// TIA Portal V17 export
// export: Created 2024-08-29T18:23:45.9111074Z, ExportSetting WithDefaults, DisplayName Totally Integrated Automation Portal, DisplayVersion V17 Update 7, DisplayName TIA Portal Openness, DisplayVersion V17 Update 7, DisplayName TIA Portal Version Control Interface, DisplayVersion V17, DisplayName SINAMICS Startdrive Advanced, DisplayVersion V17 SP2, DisplayName SINAMICS Startdrive G110M, G120, G120C, G120D, G120P, G115D, DisplayVersion V17 SP2, DisplayName SINAMICS Startdrive G130, G150, S120, S150, SINAMICS MV, S210, DisplayVersion V17 SP2, DisplayName STEP 7 Professional, DisplayVersion V17 Update 7, DisplayName STEP 7 Safety, DisplayVersion V17 Update 6, DisplayName WinCC Advanced / Unified PC, DisplayVersion V17 Update 7
FUNCTION "stationAlarms" : Void   // FC2, LAD
{ S7_Optimized_Access := 'TRUE' }
VERSION : 0.1
// stored: AutoNumber true, IsIECCheckEnabled false, SetENOAutomatically false, UDAEnableTagReadback false
   VAR_TEMP
      visualizationDefault : Bool;
   END_VAR
   VAR_TEMP   // added for the SCL form of the ladder/FBD networks
      _w1 : Bool;
      _w2 : Bool;
      _w3 : Bool;
      _w4 : Bool;
      _w5 : Bool;
   END_VAR
BEGIN

REGION Network 1: Visualization Defaults
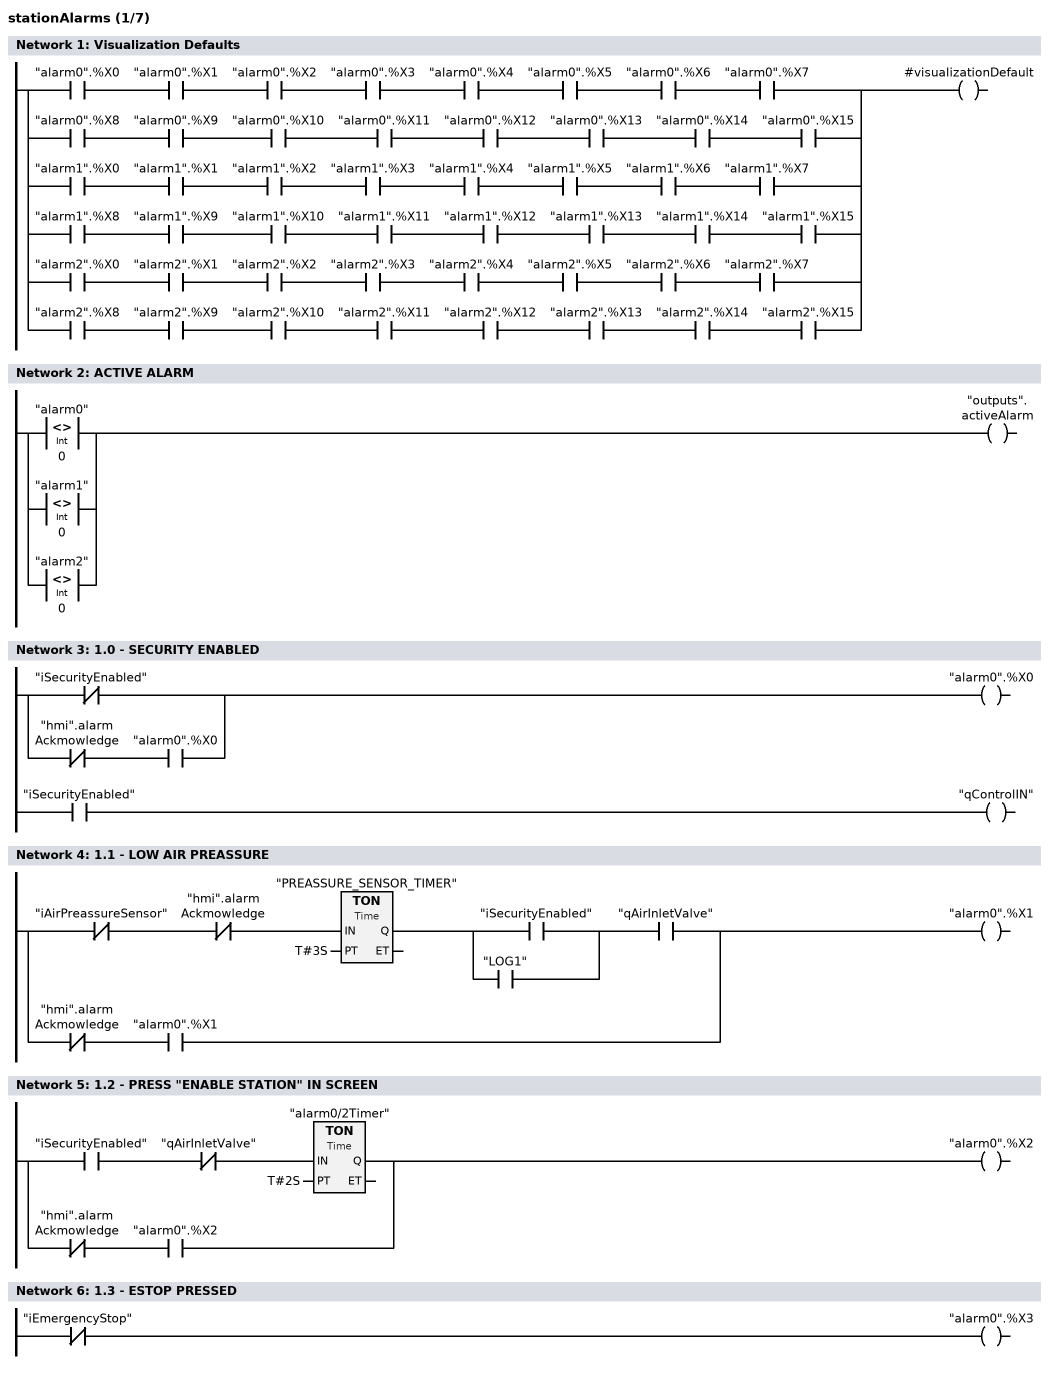
   RUNG wire#powerrail
      Contact( "alarm0".%X0 )
      Contact( "alarm0".%X1 )
      Contact( "alarm0".%X2 )
      Contact( "alarm0".%X3 )
      Contact( "alarm0".%X4 )
      Contact( "alarm0".%X5 )
      Contact( "alarm0".%X6 )
      Contact( "alarm0".%X7 )
      wire#w1
      Coil( #visualizationDefault )
   END_RUNG
   RUNG wire#powerrail
      Contact( "alarm0".%X8 )
      Contact( "alarm0".%X9 )
      Contact( "alarm0".%X10 )
      Contact( "alarm0".%X11 )
      Contact( "alarm0".%X12 )
      Contact( "alarm0".%X13 )
      Contact( "alarm0".%X14 )
      Contact( "alarm0".%X15 )
   END_RUNG wire#w1
   RUNG wire#powerrail
      Contact( "alarm1".%X0 )
      Contact( "alarm1".%X1 )
      Contact( "alarm1".%X2 )
      Contact( "alarm1".%X3 )
      Contact( "alarm1".%X4 )
      Contact( "alarm1".%X5 )
      Contact( "alarm1".%X6 )
      Contact( "alarm1".%X7 )
   END_RUNG wire#w1
   RUNG wire#powerrail
      Contact( "alarm1".%X8 )
      Contact( "alarm1".%X9 )
      Contact( "alarm1".%X10 )
      Contact( "alarm1".%X11 )
      Contact( "alarm1".%X12 )
      Contact( "alarm1".%X13 )
      Contact( "alarm1".%X14 )
      Contact( "alarm1".%X15 )
   END_RUNG wire#w1
   RUNG wire#powerrail
      Contact( "alarm2".%X0 )
      Contact( "alarm2".%X1 )
      Contact( "alarm2".%X2 )
      Contact( "alarm2".%X3 )
      Contact( "alarm2".%X4 )
      Contact( "alarm2".%X5 )
      Contact( "alarm2".%X6 )
      Contact( "alarm2".%X7 )
   END_RUNG wire#w1
   RUNG wire#powerrail
      Contact( "alarm2".%X8 )
      Contact( "alarm2".%X9 )
      Contact( "alarm2".%X10 )
      Contact( "alarm2".%X11 )
      Contact( "alarm2".%X12 )
      Contact( "alarm2".%X13 )
      Contact( "alarm2".%X14 )
      Contact( "alarm2".%X15 )
   END_RUNG wire#w1
   // the same network as SCL:
   #visualizationDefault := ("alarm0".%X0 AND "alarm0".%X1 AND "alarm0".%X2 AND "alarm0".%X3 AND "alarm0".%X4 AND "alarm0".%X5 AND "alarm0".%X6 AND "alarm0".%X7) OR ("alarm0".%X8 AND "alarm0".%X9 AND "alarm0".%X10 AND "alarm0".%X11 AND "alarm0".%X12 AND "alarm0".%X13 AND "alarm0".%X14 AND "alarm0".%X15) OR ("alarm1".%X0 AND "alarm1".%X1 AND "alarm1".%X2 AND "alarm1".%X3 AND "alarm1".%X4 AND "alarm1".%X5 AND "alarm1".%X6 AND "alarm1".%X7) OR ("alarm1".%X8 AND "alarm1".%X9 AND "alarm1".%X10 AND "alarm1".%X11 AND "alarm1".%X12 AND "alarm1".%X13 AND "alarm1".%X14 AND "alarm1".%X15) OR ("alarm2".%X0 AND "alarm2".%X1 AND "alarm2".%X2 AND "alarm2".%X3 AND "alarm2".%X4 AND "alarm2".%X5 AND "alarm2".%X6 AND "alarm2".%X7) OR ("alarm2".%X8 AND "alarm2".%X9 AND "alarm2".%X10 AND "alarm2".%X11 AND "alarm2".%X12 AND "alarm2".%X13 AND "alarm2".%X14 AND "alarm2".%X15);
END_REGION

REGION Network 2: ACTIVE ALARM
   RUNG wire#powerrail
      { S7_Templates := "SrcType := Int" } NE_Contact(in1 := "alarm0", in2 := 0)
      wire#w1
      Coil( "outputs".activeAlarm )
   END_RUNG
   RUNG wire#powerrail
      { S7_Templates := "SrcType := Int" } NE_Contact(in1 := "alarm1", in2 := 0)
   END_RUNG wire#w1
   RUNG wire#powerrail
      { S7_Templates := "SrcType := Int" } NE_Contact(in1 := "alarm2", in2 := 0)
   END_RUNG wire#w1
   // the same network as SCL:
   "outputs".activeAlarm := ("alarm0" <> 0) OR ("alarm1" <> 0) OR ("alarm2" <> 0);
END_REGION

REGION Network 3: 1.0 - SECURITY ENABLED
   RUNG wire#powerrail
      I_Contact( "iSecurityEnabled" )
      wire#w1
      Coil( "alarm0".%X0 )
   END_RUNG
   RUNG wire#powerrail
      I_Contact( "hmi".alarmAckmowledge )
      Contact( "alarm0".%X0 )
   END_RUNG wire#w1
   RUNG wire#powerrail
      Contact( "iSecurityEnabled" )
      Coil( "qControlIN" )
   END_RUNG
   // the same network as SCL:
   "alarm0".%X0 := NOT "iSecurityEnabled" OR (NOT "hmi".alarmAckmowledge AND "alarm0".%X0);
   "qControlIN" := "iSecurityEnabled";
END_REGION

REGION Network 4: 1.1 - LOW AIR PREASSURE
   RUNG wire#powerrail
      I_Contact( "iAirPreassureSensor" )
      I_Contact( "hmi".alarmAckmowledge )
      { S7_Templates := "time_type := Time" } "PREASSURE_SENSOR_TIMER".TON(pt := T#3S, et =>)
      wire#w1
      Contact( "iSecurityEnabled" )
      wire#w2
      Contact( "qAirInletValve" )
      wire#w3
      Coil( "alarm0".%X1 )
   END_RUNG
   RUNG wire#w1
      Contact( "LOG1" )
   END_RUNG wire#w2
   RUNG wire#powerrail
      I_Contact( "hmi".alarmAckmowledge )
      Contact( "alarm0".%X1 )
   END_RUNG wire#w3
   // the same network as SCL:
   "PREASSURE_SENSOR_TIMER".TON(IN := NOT "iAirPreassureSensor" AND NOT "hmi".alarmAckmowledge, PT := T#3S);
   "alarm0".%X1 := ("PREASSURE_SENSOR_TIMER".Q AND ("iSecurityEnabled" OR "LOG1") AND "qAirInletValve") OR (NOT "hmi".alarmAckmowledge AND "alarm0".%X1);
END_REGION

REGION Network 5: 1.2 - PRESS "ENABLE STATION" IN SCREEN
   RUNG wire#powerrail
      Contact( "iSecurityEnabled" )
      I_Contact( "qAirInletValve" )
      { S7_Templates := "time_type := Time" } "alarm0/2Timer".TON(pt := T#2S, et =>)
      wire#w1
      Coil( "alarm0".%X2 )
   END_RUNG
   RUNG wire#powerrail
      I_Contact( "hmi".alarmAckmowledge )
      Contact( "alarm0".%X2 )
   END_RUNG wire#w1
   // the same network as SCL:
   "alarm0/2Timer".TON(IN := "iSecurityEnabled" AND NOT "qAirInletValve", PT := T#2S);
   "alarm0".%X2 := "alarm0/2Timer".Q OR (NOT "hmi".alarmAckmowledge AND "alarm0".%X2);
END_REGION

REGION Network 6: 1.3 - ESTOP PRESSED
   RUNG wire#powerrail
      I_Contact( "iEmergencyStop" )
      Coil( "alarm0".%X3 )
   END_RUNG
   // the same network as SCL:
   "alarm0".%X3 := NOT "iEmergencyStop";
END_REGION

REGION Network 7: 1.4 - MANUAL COMMAND OUT OF MANUAL MODE
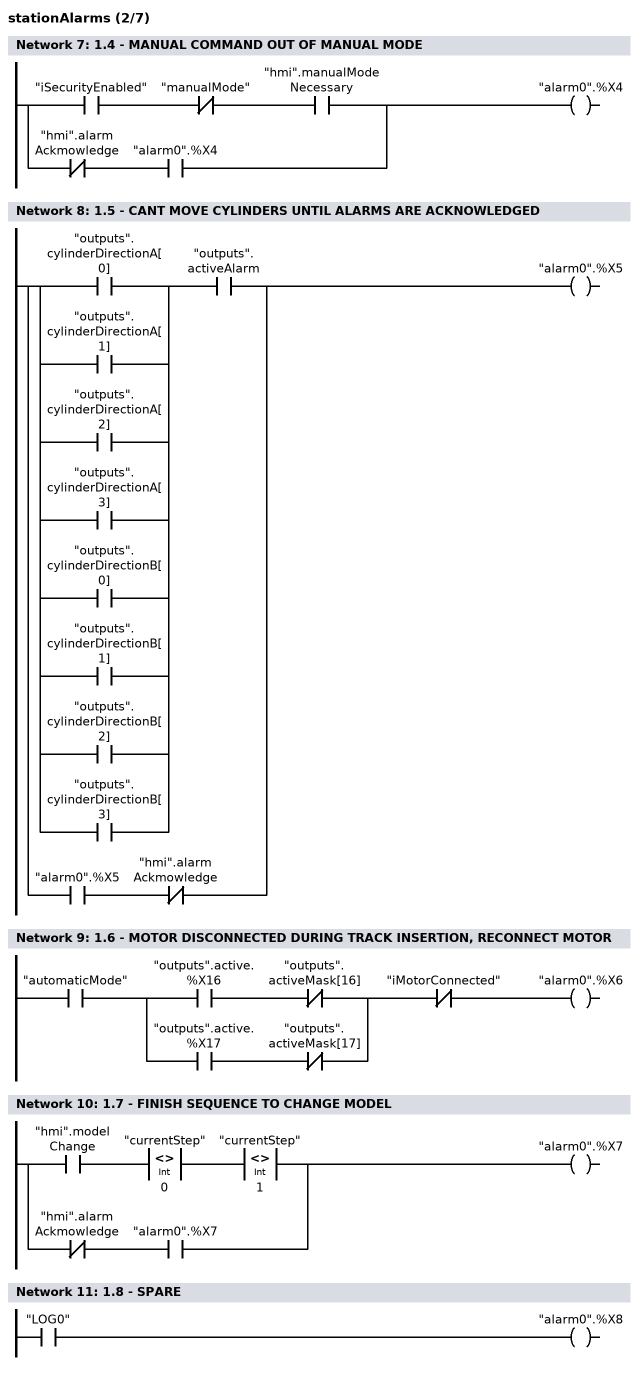
   RUNG wire#powerrail
      Contact( "iSecurityEnabled" )
      I_Contact( "manualMode" )
      Contact( "hmi".manualModeNecessary )
      wire#w1
      Coil( "alarm0".%X4 )
   END_RUNG
   RUNG wire#powerrail
      I_Contact( "hmi".alarmAckmowledge )
      Contact( "alarm0".%X4 )
   END_RUNG wire#w1
   // the same network as SCL:
   "alarm0".%X4 := ("iSecurityEnabled" AND NOT "manualMode" AND "hmi".manualModeNecessary) OR (NOT "hmi".alarmAckmowledge AND "alarm0".%X4);
END_REGION

REGION Network 8: 1.5 - CANT MOVE CYLINDERS UNTIL ALARMS ARE ACKNOWLEDGED
   RUNG wire#powerrail
      Contact( "outputs".cylinderDirectionA[0] )
      wire#w1
      Contact( "outputs".activeAlarm )
      wire#w2
      Coil( "alarm0".%X5 )
   END_RUNG
   RUNG wire#powerrail
      Contact( "outputs".cylinderDirectionA[1] )
   END_RUNG wire#w1
   RUNG wire#powerrail
      Contact( "outputs".cylinderDirectionA[2] )
   END_RUNG wire#w1
   RUNG wire#powerrail
      Contact( "outputs".cylinderDirectionA[3] )
   END_RUNG wire#w1
   RUNG wire#powerrail
      Contact( "outputs".cylinderDirectionB[0] )
   END_RUNG wire#w1
   RUNG wire#powerrail
      Contact( "outputs".cylinderDirectionB[1] )
   END_RUNG wire#w1
   RUNG wire#powerrail
      Contact( "outputs".cylinderDirectionB[2] )
   END_RUNG wire#w1
   RUNG wire#powerrail
      Contact( "outputs".cylinderDirectionB[3] )
   END_RUNG wire#w1
   RUNG wire#powerrail
      Contact( "alarm0".%X5 )
      I_Contact( "hmi".alarmAckmowledge )
   END_RUNG wire#w2
   // the same network as SCL:
   "alarm0".%X5 := (("outputs".cylinderDirectionA[0] OR "outputs".cylinderDirectionA[1] OR "outputs".cylinderDirectionA[2] OR "outputs".cylinderDirectionA[3] OR "outputs".cylinderDirectionB[0] OR "outputs".cylinderDirectionB[1] OR "outputs".cylinderDirectionB[2] OR "outputs".cylinderDirectionB[3]) AND "outputs".activeAlarm) OR ("alarm0".%X5 AND NOT "hmi".alarmAckmowledge);
END_REGION

REGION Network 9: 1.6 - MOTOR DISCONNECTED DURING TRACK INSERTION, RECONNECT MOTOR
   RUNG wire#powerrail
      Contact( "automaticMode" )
      wire#w1
      Contact( "outputs".active.%X16 )
      I_Contact( "outputs".activeMask[16] )
      wire#w2
      I_Contact( "iMotorConnected" )
      Coil( "alarm0".%X6 )
   END_RUNG
   RUNG wire#w1
      Contact( "outputs".active.%X17 )
      I_Contact( "outputs".activeMask[17] )
   END_RUNG wire#w2
   // the same network as SCL:
   "alarm0".%X6 := "automaticMode" AND (("outputs".active.%X16 AND NOT "outputs".activeMask[16]) OR ("outputs".active.%X17 AND NOT "outputs".activeMask[17])) AND NOT "iMotorConnected";
END_REGION

REGION Network 10: 1.7 - FINISH SEQUENCE TO CHANGE MODEL
   RUNG wire#powerrail
      Contact( "hmi".modelChange )
      { S7_Templates := "SrcType := Int" } NE_Contact(in1 := "currentStep", in2 := 0)
      { S7_Templates := "SrcType := Int" } NE_Contact(in1 := "currentStep", in2 := 1)
      wire#w1
      Coil( "alarm0".%X7 )
   END_RUNG
   RUNG wire#powerrail
      I_Contact( "hmi".alarmAckmowledge )
      Contact( "alarm0".%X7 )
   END_RUNG wire#w1
   // the same network as SCL:
   "alarm0".%X7 := ("hmi".modelChange AND ("currentStep" <> 0) AND ("currentStep" <> 1)) OR (NOT "hmi".alarmAckmowledge AND "alarm0".%X7);
END_REGION

REGION Network 11: 1.8 - SPARE
   RUNG wire#powerrail
      Contact( "LOG0" )
      Coil( "alarm0".%X8 )
   END_RUNG
   // the same network as SCL:
   "alarm0".%X8 := "LOG0";
END_REGION

REGION Network 12: 1.9 - WRONG TAG
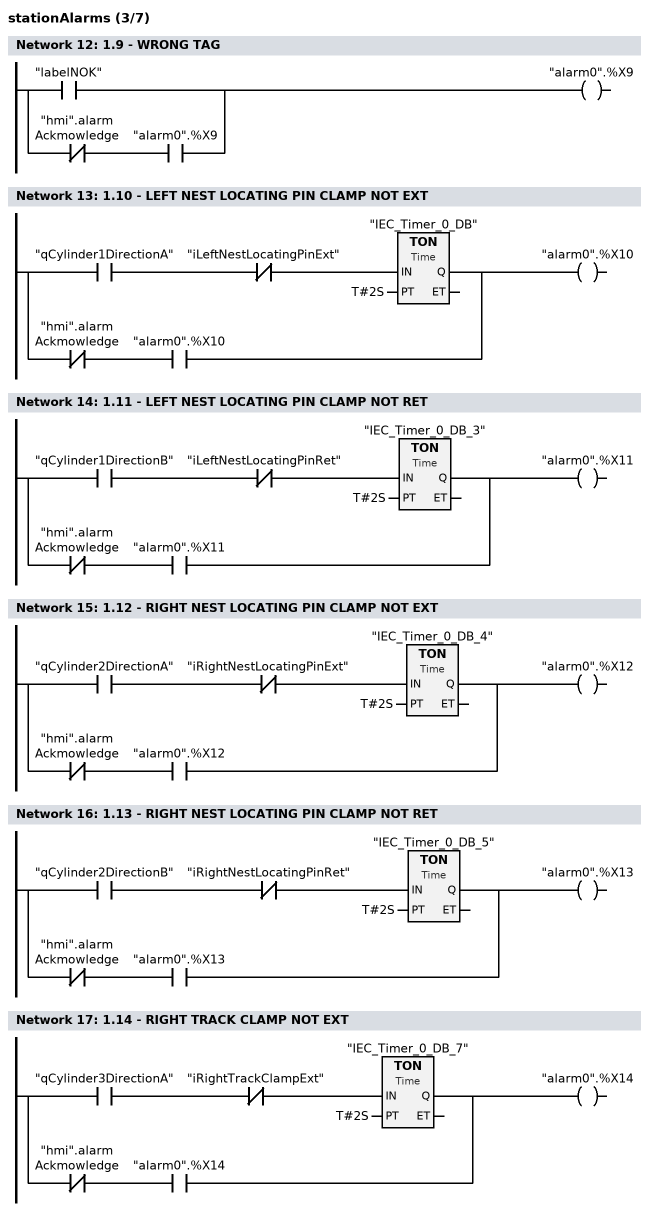
   RUNG wire#powerrail
      Contact( "labelNOK" )
      wire#w1
      Coil( "alarm0".%X9 )
   END_RUNG
   RUNG wire#powerrail
      I_Contact( "hmi".alarmAckmowledge )
      Contact( "alarm0".%X9 )
   END_RUNG wire#w1
   // the same network as SCL:
   "alarm0".%X9 := "labelNOK" OR (NOT "hmi".alarmAckmowledge AND "alarm0".%X9);
END_REGION

REGION Network 13: 1.10 - LEFT NEST LOCATING PIN CLAMP NOT EXT
   RUNG wire#powerrail
      Contact( "qCylinder1DirectionA" )
      I_Contact( "iLeftNestLocatingPinExt" )
      { S7_Templates := "time_type := Time" } "IEC_Timer_0_DB".TON(pt := T#2S, et =>)
      wire#w1
      Coil( "alarm0".%X10 )
   END_RUNG
   RUNG wire#powerrail
      I_Contact( "hmi".alarmAckmowledge )
      Contact( "alarm0".%X10 )
   END_RUNG wire#w1
   // the same network as SCL:
   "IEC_Timer_0_DB".TON(IN := "qCylinder1DirectionA" AND NOT "iLeftNestLocatingPinExt", PT := T#2S);
   "alarm0".%X10 := "IEC_Timer_0_DB".Q OR (NOT "hmi".alarmAckmowledge AND "alarm0".%X10);
END_REGION

REGION Network 14: 1.11 - LEFT NEST LOCATING PIN CLAMP NOT RET
   RUNG wire#powerrail
      Contact( "qCylinder1DirectionB" )
      I_Contact( "iLeftNestLocatingPinRet" )
      { S7_Templates := "time_type := Time" } "IEC_Timer_0_DB_3".TON(pt := T#2S, et =>)
      wire#w1
      Coil( "alarm0".%X11 )
   END_RUNG
   RUNG wire#powerrail
      I_Contact( "hmi".alarmAckmowledge )
      Contact( "alarm0".%X11 )
   END_RUNG wire#w1
   // the same network as SCL:
   "IEC_Timer_0_DB_3".TON(IN := "qCylinder1DirectionB" AND NOT "iLeftNestLocatingPinRet", PT := T#2S);
   "alarm0".%X11 := "IEC_Timer_0_DB_3".Q OR (NOT "hmi".alarmAckmowledge AND "alarm0".%X11);
END_REGION

REGION Network 15: 1.12 - RIGHT NEST LOCATING PIN CLAMP NOT EXT
   RUNG wire#powerrail
      Contact( "qCylinder2DirectionA" )
      I_Contact( "iRightNestLocatingPinExt" )
      { S7_Templates := "time_type := Time" } "IEC_Timer_0_DB_4".TON(pt := T#2S, et =>)
      wire#w1
      Coil( "alarm0".%X12 )
   END_RUNG
   RUNG wire#powerrail
      I_Contact( "hmi".alarmAckmowledge )
      Contact( "alarm0".%X12 )
   END_RUNG wire#w1
   // the same network as SCL:
   "IEC_Timer_0_DB_4".TON(IN := "qCylinder2DirectionA" AND NOT "iRightNestLocatingPinExt", PT := T#2S);
   "alarm0".%X12 := "IEC_Timer_0_DB_4".Q OR (NOT "hmi".alarmAckmowledge AND "alarm0".%X12);
END_REGION

REGION Network 16: 1.13 - RIGHT NEST LOCATING PIN CLAMP NOT RET
   RUNG wire#powerrail
      Contact( "qCylinder2DirectionB" )
      I_Contact( "iRightNestLocatingPinRet" )
      { S7_Templates := "time_type := Time" } "IEC_Timer_0_DB_5".TON(pt := T#2S, et =>)
      wire#w1
      Coil( "alarm0".%X13 )
   END_RUNG
   RUNG wire#powerrail
      I_Contact( "hmi".alarmAckmowledge )
      Contact( "alarm0".%X13 )
   END_RUNG wire#w1
   // the same network as SCL:
   "IEC_Timer_0_DB_5".TON(IN := "qCylinder2DirectionB" AND NOT "iRightNestLocatingPinRet", PT := T#2S);
   "alarm0".%X13 := "IEC_Timer_0_DB_5".Q OR (NOT "hmi".alarmAckmowledge AND "alarm0".%X13);
END_REGION

REGION Network 17: 1.14 - RIGHT TRACK CLAMP NOT EXT
   RUNG wire#powerrail
      Contact( "qCylinder3DirectionA" )
      I_Contact( "iRightTrackClampExt" )
      { S7_Templates := "time_type := Time" } "IEC_Timer_0_DB_7".TON(pt := T#2S, et =>)
      wire#w1
      Coil( "alarm0".%X14 )
   END_RUNG
   RUNG wire#powerrail
      I_Contact( "hmi".alarmAckmowledge )
      Contact( "alarm0".%X14 )
   END_RUNG wire#w1
   // the same network as SCL:
   "IEC_Timer_0_DB_7".TON(IN := "qCylinder3DirectionA" AND NOT "iRightTrackClampExt", PT := T#2S);
   "alarm0".%X14 := "IEC_Timer_0_DB_7".Q OR (NOT "hmi".alarmAckmowledge AND "alarm0".%X14);
END_REGION

REGION Network 18: 1.15 - RIGHT TRACK CLAMP NOT RET
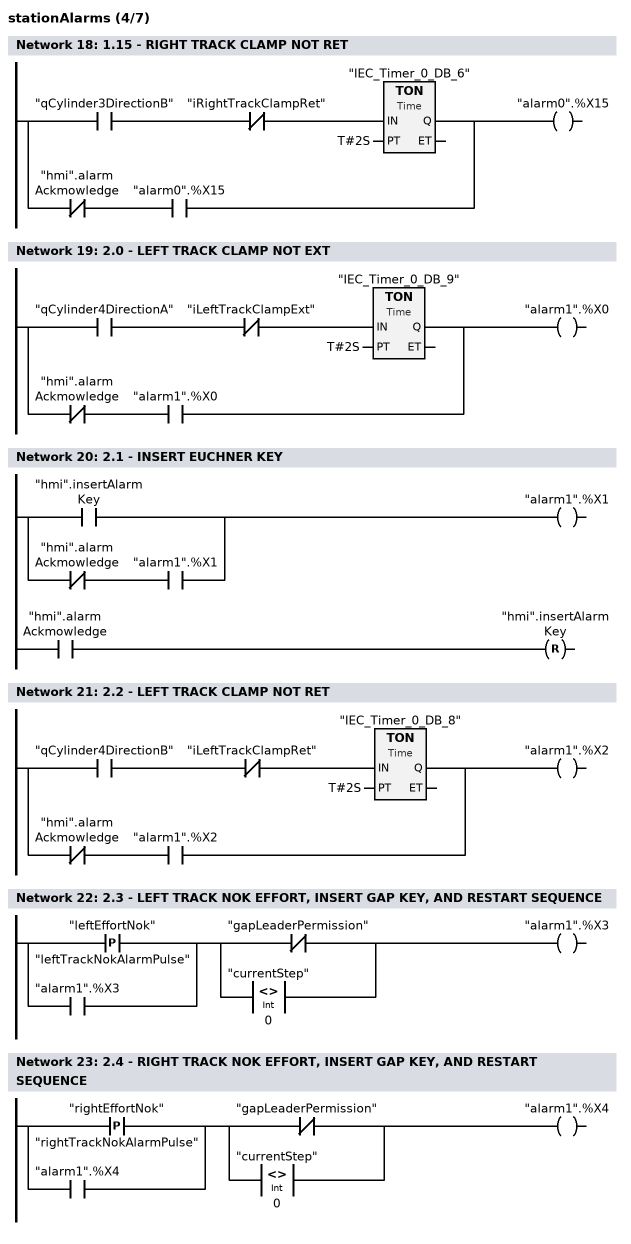
   RUNG wire#powerrail
      Contact( "qCylinder3DirectionB" )
      I_Contact( "iRightTrackClampRet" )
      { S7_Templates := "time_type := Time" } "IEC_Timer_0_DB_6".TON(pt := T#2S, et =>)
      wire#w1
      Coil( "alarm0".%X15 )
   END_RUNG
   RUNG wire#powerrail
      I_Contact( "hmi".alarmAckmowledge )
      Contact( "alarm0".%X15 )
   END_RUNG wire#w1
   // the same network as SCL:
   "IEC_Timer_0_DB_6".TON(IN := "qCylinder3DirectionB" AND NOT "iRightTrackClampRet", PT := T#2S);
   "alarm0".%X15 := "IEC_Timer_0_DB_6".Q OR (NOT "hmi".alarmAckmowledge AND "alarm0".%X15);
END_REGION

REGION Network 19: 2.0 - LEFT TRACK CLAMP NOT EXT
   RUNG wire#powerrail
      Contact( "qCylinder4DirectionA" )
      I_Contact( "iLeftTrackClampExt" )
      { S7_Templates := "time_type := Time" } "IEC_Timer_0_DB_9".TON(pt := T#2S, et =>)
      wire#w1
      Coil( "alarm1".%X0 )
   END_RUNG
   RUNG wire#powerrail
      I_Contact( "hmi".alarmAckmowledge )
      Contact( "alarm1".%X0 )
   END_RUNG wire#w1
   // the same network as SCL:
   "IEC_Timer_0_DB_9".TON(IN := "qCylinder4DirectionA" AND NOT "iLeftTrackClampExt", PT := T#2S);
   "alarm1".%X0 := "IEC_Timer_0_DB_9".Q OR (NOT "hmi".alarmAckmowledge AND "alarm1".%X0);
END_REGION

REGION Network 20: 2.1 - INSERT EUCHNER KEY
   RUNG wire#powerrail
      Contact( "hmi".insertAlarmKey )
      wire#w1
      Coil( "alarm1".%X1 )
   END_RUNG
   RUNG wire#powerrail
      I_Contact( "hmi".alarmAckmowledge )
      Contact( "alarm1".%X1 )
   END_RUNG wire#w1
   RUNG wire#powerrail
      Contact( "hmi".alarmAckmowledge )
      R_Coil( "hmi".insertAlarmKey )
   END_RUNG
   // the same network as SCL:
   "alarm1".%X1 := "hmi".insertAlarmKey OR (NOT "hmi".alarmAckmowledge AND "alarm1".%X1);
   IF "hmi".alarmAckmowledge THEN "hmi".insertAlarmKey := FALSE; END_IF;
END_REGION

REGION Network 21: 2.2 - LEFT TRACK CLAMP NOT RET
   RUNG wire#powerrail
      Contact( "qCylinder4DirectionB" )
      I_Contact( "iLeftTrackClampRet" )
      { S7_Templates := "time_type := Time" } "IEC_Timer_0_DB_8".TON(pt := T#2S, et =>)
      wire#w1
      Coil( "alarm1".%X2 )
   END_RUNG
   RUNG wire#powerrail
      I_Contact( "hmi".alarmAckmowledge )
      Contact( "alarm1".%X2 )
   END_RUNG wire#w1
   // the same network as SCL:
   "IEC_Timer_0_DB_8".TON(IN := "qCylinder4DirectionB" AND NOT "iLeftTrackClampRet", PT := T#2S);
   "alarm1".%X2 := "IEC_Timer_0_DB_8".Q OR (NOT "hmi".alarmAckmowledge AND "alarm1".%X2);
END_REGION

REGION Network 22: 2.3 - LEFT TRACK NOK EFFORT, INSERT GAP KEY, AND RESTART SEQUENCE
   RUNG wire#powerrail
      P_Contact(operand := "leftEffortNok", bit := "leftTrackNokAlarmPulse")
      wire#w1
      I_Contact( "gapLeaderPermission" )
      wire#w2
      Coil( "alarm1".%X3 )
   END_RUNG
   RUNG wire#powerrail
      Contact( "alarm1".%X3 )
   END_RUNG wire#w1
   RUNG wire#w1
      { S7_Templates := "SrcType := Int" } NE_Contact(in1 := "currentStep", in2 := 0)
   END_RUNG wire#w2
   // the same network as SCL:
   #_w1 := "leftEffortNok" AND NOT "leftTrackNokAlarmPulse";   // rising edge of "leftEffortNok"
   "leftTrackNokAlarmPulse" := "leftEffortNok";
   "alarm1".%X3 := (#_w1 OR "alarm1".%X3) AND (NOT "gapLeaderPermission" OR ("currentStep" <> 0));
END_REGION

REGION Network 23: 2.4 - RIGHT TRACK NOK EFFORT, INSERT GAP KEY, AND RESTART SEQUENCE
   RUNG wire#powerrail
      P_Contact(operand := "rightEffortNok", bit := "rightTrackNokAlarmPulse")
      wire#w1
      I_Contact( "gapLeaderPermission" )
      wire#w2
      Coil( "alarm1".%X4 )
   END_RUNG
   RUNG wire#powerrail
      Contact( "alarm1".%X4 )
   END_RUNG wire#w1
   RUNG wire#w1
      { S7_Templates := "SrcType := Int" } NE_Contact(in1 := "currentStep", in2 := 0)
   END_RUNG wire#w2
   // the same network as SCL:
   #_w1 := "rightEffortNok" AND NOT "rightTrackNokAlarmPulse";   // rising edge of "rightEffortNok"
   "rightTrackNokAlarmPulse" := "rightEffortNok";
   "alarm1".%X4 := (#_w1 OR "alarm1".%X4) AND (NOT "gapLeaderPermission" OR ("currentStep" <> 0));
END_REGION

REGION Network 24: 2.5 - SELECT MODELTO RUN
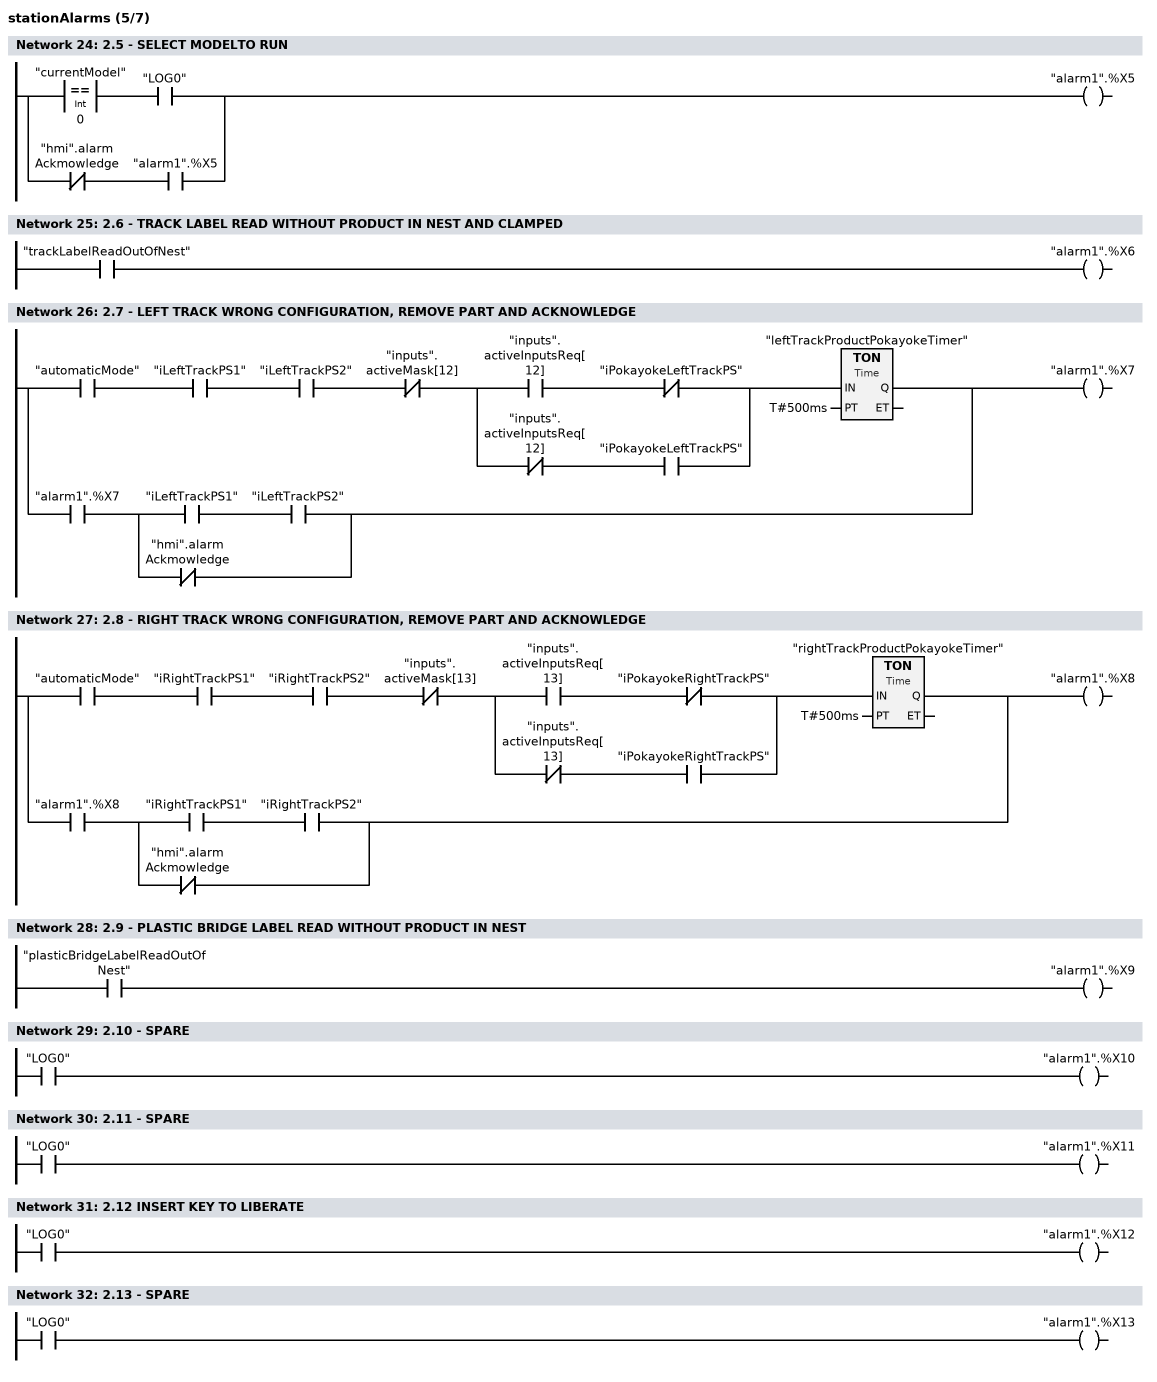
   RUNG wire#powerrail
      { S7_Templates := "SrcType := Int" } EQ_Contact(in1 := "currentModel", in2 := 0)
      Contact( "LOG0" )
      wire#w1
      Coil( "alarm1".%X5 )
   END_RUNG
   RUNG wire#powerrail
      I_Contact( "hmi".alarmAckmowledge )
      Contact( "alarm1".%X5 )
   END_RUNG wire#w1
   // the same network as SCL:
   "alarm1".%X5 := (("currentModel" = 0) AND "LOG0") OR (NOT "hmi".alarmAckmowledge AND "alarm1".%X5);
END_REGION

REGION Network 25: 2.6 - TRACK LABEL READ WITHOUT PRODUCT IN NEST AND CLAMPED
   RUNG wire#powerrail
      Contact( "trackLabelReadOutOfNest" )
      Coil( "alarm1".%X6 )
   END_RUNG
   // the same network as SCL:
   "alarm1".%X6 := "trackLabelReadOutOfNest";
END_REGION

REGION Network 26: 2.7 - LEFT TRACK WRONG CONFIGURATION, REMOVE PART AND ACKNOWLEDGE
   RUNG wire#powerrail
      Contact( "automaticMode" )
      Contact( "iLeftTrackPS1" )
      Contact( "iLeftTrackPS2" )
      I_Contact( "inputs".activeMask[12] )
      wire#w1
      Contact( "inputs".activeInputsReq[12] )
      I_Contact( "iPokayokeLeftTrackPS" )
      wire#w2
      { S7_Templates := "time_type := Time" } "leftTrackProductPokayokeTimer".TON(pt := T#500ms, et =>)
      wire#w3
      Coil( "alarm1".%X7 )
   END_RUNG
   RUNG wire#w1
      I_Contact( "inputs".activeInputsReq[12] )
      Contact( "iPokayokeLeftTrackPS" )
   END_RUNG wire#w2
   RUNG wire#powerrail
      Contact( "alarm1".%X7 )
      wire#w4
      Contact( "iLeftTrackPS1" )
      Contact( "iLeftTrackPS2" )
   END_RUNG wire#w3
   RUNG wire#w4
      I_Contact( "hmi".alarmAckmowledge )
   END_RUNG wire#w3
   // the same network as SCL:
   "leftTrackProductPokayokeTimer".TON(IN := "automaticMode" AND "iLeftTrackPS1" AND "iLeftTrackPS2" AND NOT "inputs".activeMask[12] AND (("inputs".activeInputsReq[12] AND NOT "iPokayokeLeftTrackPS") OR (NOT "inputs".activeInputsReq[12] AND "iPokayokeLeftTrackPS")),
                           PT := T#500ms);
   "alarm1".%X7 := "leftTrackProductPokayokeTimer".Q OR ("alarm1".%X7 AND (("iLeftTrackPS1" AND "iLeftTrackPS2") OR NOT "hmi".alarmAckmowledge));
END_REGION

REGION Network 27: 2.8 - RIGHT TRACK WRONG CONFIGURATION, REMOVE PART AND ACKNOWLEDGE
   RUNG wire#powerrail
      Contact( "automaticMode" )
      Contact( "iRightTrackPS1" )
      Contact( "iRightTrackPS2" )
      I_Contact( "inputs".activeMask[13] )
      wire#w1
      Contact( "inputs".activeInputsReq[13] )
      I_Contact( "iPokayokeRightTrackPS" )
      wire#w2
      { S7_Templates := "time_type := Time" } "rightTrackProductPokayokeTimer".TON(pt := T#500ms, et =>)
      wire#w3
      Coil( "alarm1".%X8 )
   END_RUNG
   RUNG wire#w1
      I_Contact( "inputs".activeInputsReq[13] )
      Contact( "iPokayokeRightTrackPS" )
   END_RUNG wire#w2
   RUNG wire#powerrail
      Contact( "alarm1".%X8 )
      wire#w4
      Contact( "iRightTrackPS1" )
      Contact( "iRightTrackPS2" )
   END_RUNG wire#w3
   RUNG wire#w4
      I_Contact( "hmi".alarmAckmowledge )
   END_RUNG wire#w3
   // the same network as SCL:
   "rightTrackProductPokayokeTimer".TON(IN := "automaticMode" AND "iRightTrackPS1" AND "iRightTrackPS2" AND NOT "inputs".activeMask[13] AND (("inputs".activeInputsReq[13] AND NOT "iPokayokeRightTrackPS") OR (NOT "inputs".activeInputsReq[13] AND "iPokayokeRightTrackPS")),
                           PT := T#500ms);
   "alarm1".%X8 := "rightTrackProductPokayokeTimer".Q OR ("alarm1".%X8 AND (("iRightTrackPS1" AND "iRightTrackPS2") OR NOT "hmi".alarmAckmowledge));
END_REGION

REGION Network 28: 2.9 - PLASTIC BRIDGE LABEL READ WITHOUT PRODUCT IN NEST
   RUNG wire#powerrail
      Contact( "plasticBridgeLabelReadOutOfNest" )
      Coil( "alarm1".%X9 )
   END_RUNG
   // the same network as SCL:
   "alarm1".%X9 := "plasticBridgeLabelReadOutOfNest";
END_REGION

REGION Network 29: 2.10 - SPARE
   RUNG wire#powerrail
      Contact( "LOG0" )
      Coil( "alarm1".%X10 )
   END_RUNG
   // the same network as SCL:
   "alarm1".%X10 := "LOG0";
END_REGION

REGION Network 30: 2.11 - SPARE
   RUNG wire#powerrail
      Contact( "LOG0" )
      Coil( "alarm1".%X11 )
   END_RUNG
   // the same network as SCL:
   "alarm1".%X11 := "LOG0";
END_REGION

REGION Network 31: 2.12 INSERT KEY TO LIBERATE
   RUNG wire#powerrail
      Contact( "LOG0" )
      Coil( "alarm1".%X12 )
   END_RUNG
   // the same network as SCL:
   "alarm1".%X12 := "LOG0";
END_REGION

REGION Network 32: 2.13 - SPARE
   RUNG wire#powerrail
      Contact( "LOG0" )
      Coil( "alarm1".%X13 )
   END_RUNG
   // the same network as SCL:
   "alarm1".%X13 := "LOG0";
END_REGION

REGION Network 33: 2.14 - SPARE
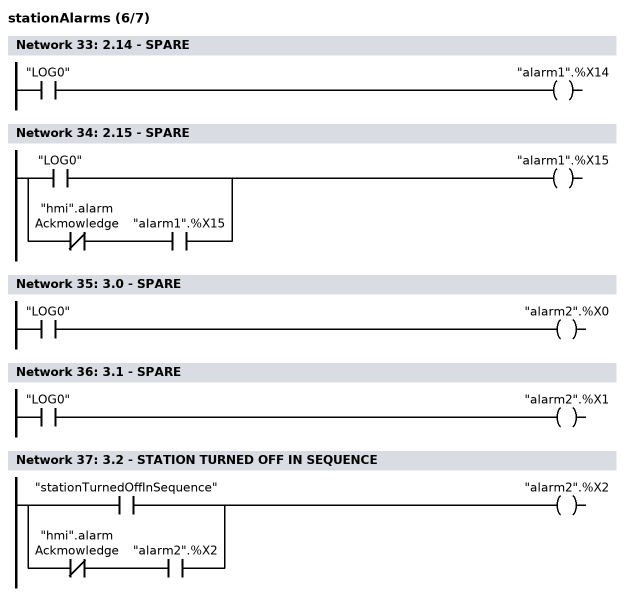
   RUNG wire#powerrail
      Contact( "LOG0" )
      Coil( "alarm1".%X14 )
   END_RUNG
   // the same network as SCL:
   "alarm1".%X14 := "LOG0";
END_REGION

REGION Network 34: 2.15 - SPARE
   RUNG wire#powerrail
      Contact( "LOG0" )
      wire#w1
      Coil( "alarm1".%X15 )
   END_RUNG
   RUNG wire#powerrail
      I_Contact( "hmi".alarmAckmowledge )
      Contact( "alarm1".%X15 )
   END_RUNG wire#w1
   // the same network as SCL:
   "alarm1".%X15 := "LOG0" OR (NOT "hmi".alarmAckmowledge AND "alarm1".%X15);
END_REGION

REGION Network 35: 3.0 - SPARE
   RUNG wire#powerrail
      Contact( "LOG0" )
      Coil( "alarm2".%X0 )
   END_RUNG
   // the same network as SCL:
   "alarm2".%X0 := "LOG0";
END_REGION

REGION Network 36: 3.1 - SPARE
   RUNG wire#powerrail
      Contact( "LOG0" )
      Coil( "alarm2".%X1 )
   END_RUNG
   // the same network as SCL:
   "alarm2".%X1 := "LOG0";
END_REGION

REGION Network 37: 3.2 - STATION TURNED OFF IN SEQUENCE
   RUNG wire#powerrail
      Contact( "stationTurnedOffInSequence" )
      wire#w1
      Coil( "alarm2".%X2 )
   END_RUNG
   RUNG wire#powerrail
      I_Contact( "hmi".alarmAckmowledge )
      Contact( "alarm2".%X2 )
   END_RUNG wire#w1
   // the same network as SCL:
   "alarm2".%X2 := "stationTurnedOffInSequence" OR (NOT "hmi".alarmAckmowledge AND "alarm2".%X2);
END_REGION

REGION Network 38: 3.3 - 3.13 COMMUNICATION ALARMS
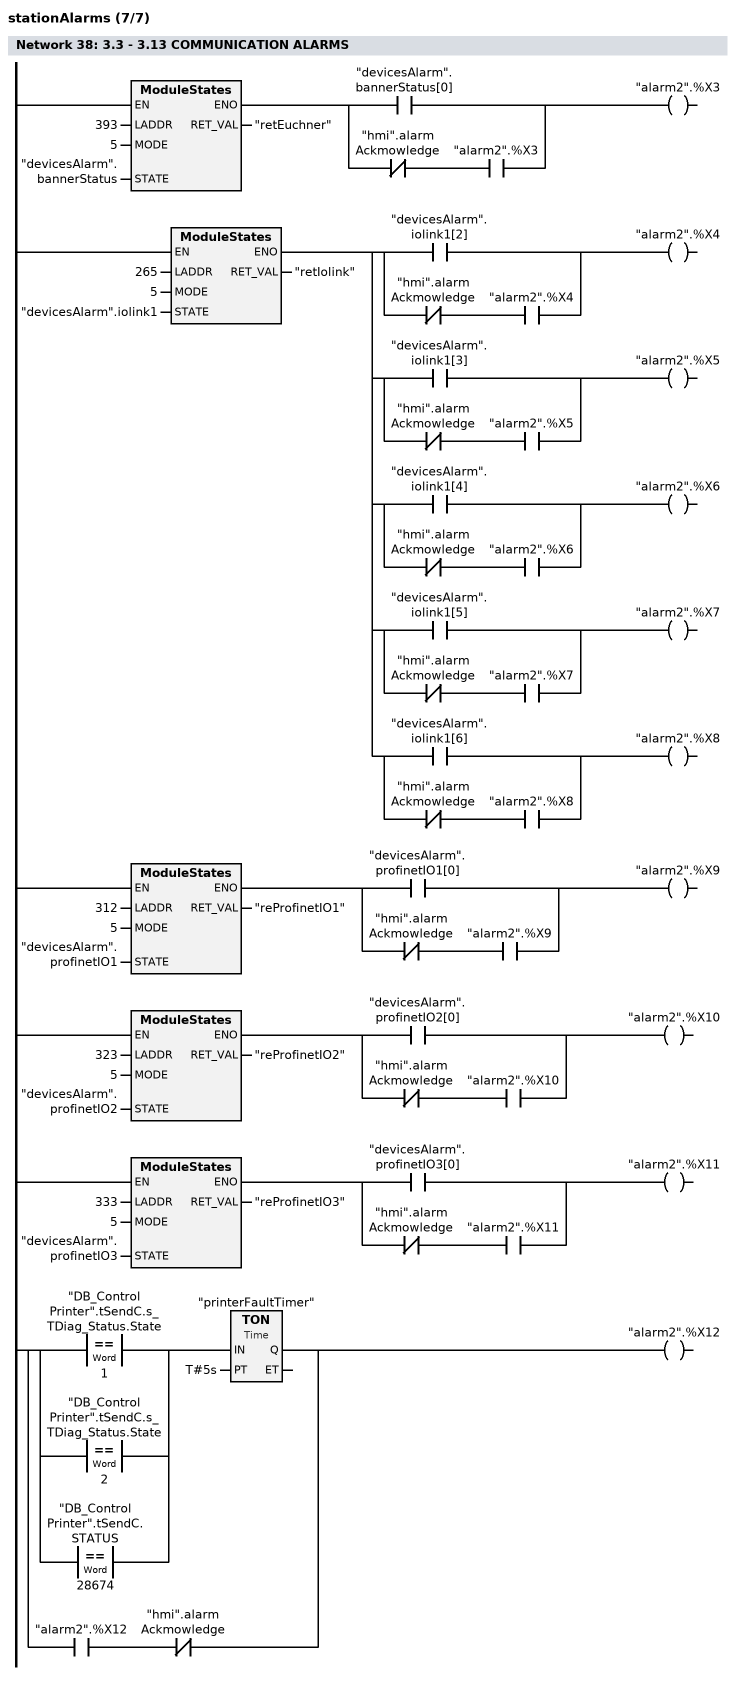
   RUNG wire#powerrail
      ModuleStates(LADDR := 393, MODE := 5, STATE := "devicesAlarm".bannerStatus, Ret_Val => "retEuchner")
      wire#w1
      Contact( "devicesAlarm".bannerStatus[0] )
      wire#w2
      Coil( "alarm2".%X3 )
   END_RUNG
   RUNG wire#w1
      I_Contact( "hmi".alarmAckmowledge )
      Contact( "alarm2".%X3 )
   END_RUNG wire#w2
   RUNG wire#powerrail
      ModuleStates(LADDR := 265, MODE := 5, STATE := "devicesAlarm".iolink1, Ret_Val => "retIolink")
      wire#w3
      Contact( "devicesAlarm".iolink1[2] )
      wire#w4
      Coil( "alarm2".%X4 )
   END_RUNG
   RUNG wire#w3
      I_Contact( "hmi".alarmAckmowledge )
      Contact( "alarm2".%X4 )
   END_RUNG wire#w4
   RUNG wire#w3
      Contact( "devicesAlarm".iolink1[3] )
      wire#w5
      Coil( "alarm2".%X5 )
   END_RUNG
   RUNG wire#w3
      I_Contact( "hmi".alarmAckmowledge )
      Contact( "alarm2".%X5 )
   END_RUNG wire#w5
   RUNG wire#w3
      Contact( "devicesAlarm".iolink1[4] )
      wire#w6
      Coil( "alarm2".%X6 )
   END_RUNG
   RUNG wire#w3
      I_Contact( "hmi".alarmAckmowledge )
      Contact( "alarm2".%X6 )
   END_RUNG wire#w6
   RUNG wire#w3
      Contact( "devicesAlarm".iolink1[5] )
      wire#w7
      Coil( "alarm2".%X7 )
   END_RUNG
   RUNG wire#w3
      I_Contact( "hmi".alarmAckmowledge )
      Contact( "alarm2".%X7 )
   END_RUNG wire#w7
   RUNG wire#w3
      Contact( "devicesAlarm".iolink1[6] )
      wire#w8
      Coil( "alarm2".%X8 )
   END_RUNG
   RUNG wire#w3
      I_Contact( "hmi".alarmAckmowledge )
      Contact( "alarm2".%X8 )
   END_RUNG wire#w8
   RUNG wire#powerrail
      ModuleStates(LADDR := 312, MODE := 5, STATE := "devicesAlarm".profinetIO1, Ret_Val => "reProfinetIO1")
      wire#w9
      Contact( "devicesAlarm".profinetIO1[0] )
      wire#w10
      Coil( "alarm2".%X9 )
   END_RUNG
   RUNG wire#w9
      I_Contact( "hmi".alarmAckmowledge )
      Contact( "alarm2".%X9 )
   END_RUNG wire#w10
   RUNG wire#powerrail
      ModuleStates(LADDR := 323, MODE := 5, STATE := "devicesAlarm".profinetIO2, Ret_Val => "reProfinetIO2")
      wire#w11
      Contact( "devicesAlarm".profinetIO2[0] )
      wire#w12
      Coil( "alarm2".%X10 )
   END_RUNG
   RUNG wire#w11
      I_Contact( "hmi".alarmAckmowledge )
      Contact( "alarm2".%X10 )
   END_RUNG wire#w12
   RUNG wire#powerrail
      ModuleStates(LADDR := 333, MODE := 5, STATE := "devicesAlarm".profinetIO3, Ret_Val => "reProfinetIO3")
      wire#w13
      Contact( "devicesAlarm".profinetIO3[0] )
      wire#w14
      Coil( "alarm2".%X11 )
   END_RUNG
   RUNG wire#w13
      I_Contact( "hmi".alarmAckmowledge )
      Contact( "alarm2".%X11 )
   END_RUNG wire#w14
   RUNG wire#powerrail
      { S7_Templates := "SrcType := Word" } EQ_Contact(in1 := "DB_ControlPrinter".tSendC.s_TDiag_Status.State, in2 := 1)
      wire#w15
      { S7_Templates := "time_type := Time" } "printerFaultTimer".TON(pt := T#5s, et =>)
      wire#w16
      Coil( "alarm2".%X12 )
   END_RUNG
   RUNG wire#powerrail
      { S7_Templates := "SrcType := Word" } EQ_Contact(in1 := "DB_ControlPrinter".tSendC.s_TDiag_Status.State, in2 := 2)
   END_RUNG wire#w15
   RUNG wire#powerrail
      { S7_Templates := "SrcType := Word" } EQ_Contact(in1 := "DB_ControlPrinter".tSendC.STATUS, in2 := 28674)
   END_RUNG wire#w15
   RUNG wire#powerrail
      Contact( "alarm2".%X12 )
      I_Contact( "hmi".alarmAckmowledge )
   END_RUNG wire#w16
   // the same network as SCL:
   "retEuchner" := ModuleStates(LADDR := 393, MODE := 5, STATE := "devicesAlarm".bannerStatus, ENO => #_w1);
   "alarm2".%X3 := #_w1 AND ("devicesAlarm".bannerStatus[0] OR (NOT "hmi".alarmAckmowledge AND "alarm2".%X3));
   "retIolink" := ModuleStates(LADDR := 265, MODE := 5, STATE := "devicesAlarm".iolink1, ENO => #_w2);
   "alarm2".%X4 := #_w2 AND ("devicesAlarm".iolink1[2] OR (NOT "hmi".alarmAckmowledge AND "alarm2".%X4));
   "alarm2".%X5 := #_w2 AND ("devicesAlarm".iolink1[3] OR (NOT "hmi".alarmAckmowledge AND "alarm2".%X5));
   "alarm2".%X6 := #_w2 AND ("devicesAlarm".iolink1[4] OR (NOT "hmi".alarmAckmowledge AND "alarm2".%X6));
   "alarm2".%X7 := #_w2 AND ("devicesAlarm".iolink1[5] OR (NOT "hmi".alarmAckmowledge AND "alarm2".%X7));
   "alarm2".%X8 := #_w2 AND ("devicesAlarm".iolink1[6] OR (NOT "hmi".alarmAckmowledge AND "alarm2".%X8));
   "reProfinetIO1" := ModuleStates(LADDR := 312, MODE := 5, STATE := "devicesAlarm".profinetIO1, ENO => #_w3);
   "alarm2".%X9 := #_w3 AND ("devicesAlarm".profinetIO1[0] OR (NOT "hmi".alarmAckmowledge AND "alarm2".%X9));
   "reProfinetIO2" := ModuleStates(LADDR := 323, MODE := 5, STATE := "devicesAlarm".profinetIO2, ENO => #_w4);
   "alarm2".%X10 := #_w4 AND ("devicesAlarm".profinetIO2[0] OR (NOT "hmi".alarmAckmowledge AND "alarm2".%X10));
   "reProfinetIO3" := ModuleStates(LADDR := 333, MODE := 5, STATE := "devicesAlarm".profinetIO3, ENO => #_w5);
   "alarm2".%X11 := #_w5 AND ("devicesAlarm".profinetIO3[0] OR (NOT "hmi".alarmAckmowledge AND "alarm2".%X11));
   "printerFaultTimer".TON(IN := ("DB_ControlPrinter".tSendC.s_TDiag_Status.State = 1) OR ("DB_ControlPrinter".tSendC.s_TDiag_Status.State = 2) OR ("DB_ControlPrinter".tSendC.STATUS = 28674),
                           PT := T#5s);
   "alarm2".%X12 := "printerFaultTimer".Q OR ("alarm2".%X12 AND NOT "hmi".alarmAckmowledge);
END_REGION
END_FUNCTION
